Staubli VAL3: HMI_setNewValue.pgx

public program HMI_setNewValue(num& x_nValue, num x_nMin, num x_nMax, num x_nX, num x_nY, string& x_sItem)
  local bool l_bOk
  local bool l_bQuit
  local string l_sMessage
begin
  call use:clear(0,13)
  do
    do
      call use:setSizeList(x_nX,x_nY-2,23,1)
      call use:listcreate("")
      call use:type(35,13,"OK")
      gotoxy(x_nX+1,x_nY-1)
      put(x_sItem)
      do
        nKey=get(x_nValue)
      until nKey==270 or nKey==278
      if x_nMin==0 and x_nMax==0
        l_bOk=true
      elseIf  x_nValue>=x_nMin and x_nValue<=x_nMax
          l_bOk=true
      else
        call language2:message(l_sMessage,38)
        popUpMsg(l_sMessage)
      endIf

    until l_bOk
    if nKey==278
      l_bQuit=true
    endIf
    call use:nullKey(nKey)
  until l_bQuit
end
